PROGRAM MAIN
VAR
END_VAR

GarageDoor();

END_PROGRAM

(* stored: Version 1.1.0.1, ProductVersion 3.1.4024.12
   POU MAIN: Id {b43837f9-e791-49bf-9c5d-58212312be3b}, SpecialFunc None *)
